// TIA Portal V19 export
TYPE "C501_STU_JPP_TYPIC"
   STRUCT
      CMD { ExternalAccessible := 'False'; ExternalVisible := 'False'; ExternalWritable := 'False'} : USInt;   // Sturing pomppaar
      VGV_LDE { ExternalAccessible := 'False'; ExternalVisible := 'False'; ExternalWritable := 'False'} : USInt;   // Vrijgave lekdetectie
      VGV_SME_L { ExternalAccessible := 'False'; ExternalVisible := 'False'; ExternalWritable := 'False'} : USInt;   // Vrijgave detectie debiet te laag
   END_STRUCT;
END_TYPE
